// TIA Portal V16 export
// export: Created 2021-07-12T14:47:18.0879408Z, ExportSetting WithDefaults, DisplayName Totally Integrated Automation Portal, DisplayVersion V16, DisplayName TIA Portal Version Control Interface, DisplayVersion V16, DisplayName TIA Portal Openness, DisplayVersion V16, DisplayName STEP 7 Professional, DisplayVersion V16, DisplayName STEP 7 Safety, DisplayVersion V16, DisplayName WinCC Professional, DisplayVersion V16
TYPE "SimaHydTO_typeHMIConnectionAdvancedAxisControlCommand"
TITLE = SimaHydTO_typeHMIConnectionAdvancedAxisControlCommand
// HMI interface: Advanced axis control
// stored: IsFailsafeCompliant false
   STRUCT
      moveRelativeExecute : Bool;   // MC_MoveRelative: Start job with a positive edge
      moveRelativeDistance : LReal;   // Distance of relative movement
      moveAbsoluteExecute : Bool;   // MC_MoveAbsolute: Start job with a positive edge
      moveAbsolutePosition : LReal;   // Target position of absolute movement
      moveAbsoluteDirection : Int := 3;   // Direction of absolute movement: 0: Positive direction / 1: Negative direction / 3: Shortest direction
      haltExecute : Bool;   // MC_Halt: Start job with a positive edge
      haltAbortAcceleration : Bool;   // Acceleration control: False: The current acceleration at the start of the job is reduced using the configured jerk. Afterwards, the deceleration builds up / True: The acceleration is set to 0.0 at the start of the job, and the deceleration immediately builds up.
      Velocity : LReal := -1.0;   // Velocity of movement
      Acceleration : LReal := -1.0;   // Acceleration of movement
      Deceleration : LReal := -1.0;   // Deceleration of movement
      Jerk : LReal := -1.0;   // Jerk of movement
   END_STRUCT;
END_TYPE
